{attribute 'qualified_only'}
VAR_GLOBAL
	VIS_SysReset		:BOOL;
END_VAR

(* stored: Version 1.1.0.1, ProductVersion 3.1.4024.12
   GVL GVL: Id {beca1180-e303-42f1-a624-fa2443fd59a6} *)
